PROGRAM MAIN
VAR
	unsorted : ARRAY [1..101] OF LREAL;
	lower: DINT;
	i: DINT;
	upper: DINT;
	rand_generator: DRAND := (Seed := 154);
END_VAR

lower := LOWER_BOUND(unsorted, 1);
upper := UPPER_BOUND(unsorted, 1);

FOR i:=lower TO upper DO
  rand_generator(Num=>unsorted[i]);
END_FOR

SortArray(target := unsorted);

FOR i:=lower TO upper DO
  rand_generator(Num=>unsorted[i]);
END_FOR


HeapSort(target := unsorted);

END_PROGRAM

(* stored: Version 1.1.0.1, ProductVersion 3.1.4026.0
   POU MAIN: Id {3ce1961a-3939-4be8-98ec-90464e47830d}, SpecialFunc None *)
